(* PLC project Topicos, Desconocido Sin nombre 1 *)
(* stored: creationDateTime 2024-03-11T19:08:26, modificationDateTime 2024-03-26T02:22:43 *)

FUNCTION_BLOCK RedPetri
  VAR_EXTERNAL
    E_0 : BOOL;
    E_1 : BOOL;
    E_2 : BOOL;
    E_3 : BOOL;
    E_4 : BOOL;
    E_5 : BOOL;
    E_6 : BOOL;
    E_7 : BOOL;
    Start_Button : BOOL;
    Stop_Button : BOOL;
    Reset_Button : BOOL;
    Blue_Product_base_Sensor : BOOL;
    Green_Product_base_Sensor : BOOL;
    Metal_Product_base_Sensor : BOOL;
    Blue_Product_base_Sensor2 : BOOL;
    Green_Product_base_Sensor_2 : BOOL;
    Metal_Product_base_Sensor2 : BOOL;
    Blue_Product_Lid_Sensor : BOOL;
    Green_Product_Lid_Sensor : BOOL;
    Metal_Product_Lid_Sensor : BOOL;
    Blue_Item_Detected_Sensor : BOOL;
    Green_Item_Detected_Sensor : BOOL;
    Metal_Item_Detected_Sensor : BOOL;
    Blue_Item_Detected_Sensor_2 : BOOL;
    Green_Item_Detected_Sensor_2 : BOOL;
    Metal_Item_Detected_Sensor_2 : BOOL;
    Blue_Stackable_Box_Sensor : BOOL;
    Green_Stackable_Box_Sensor : BOOL;
    Metal_Stackable_Box_Sensor : BOOL;
    Blue_Rotate_sensor : BOOL;
    Green_Rotate_sensor : BOOL;
    Metal_Rotate_sensor : BOOL;
    Stacker_Crane_2_Moving_X : BOOL;
    Stacker_Crane_2_Moving_Z : BOOL;
    Stacker_Crane_3_Moving_X : BOOL;
    Stacker_Crane_3_Moving_Z : BOOL;
    Stacker_Crane_4_Moving_X : BOOL;
    Stacker_Crane_4_Moving_Z : BOOL;
    Turntable_GS_0_G_Sensor : BOOL;
    Turntable_GS_90_G_Sensor : BOOL;
    Turntable_GS_Back_Sensor : BOOL;
    Turntable_GS_Front_Sensor : BOOL;
    Turntable_MS_0_G_Sensor : BOOL;
    Turntable_MS_90_G_Sensor : BOOL;
    Turntable_MS_Back_Sensor : BOOL;
    Turntable_MS_Front_Sensor : BOOL;
    Sensor_Turntable_Blue_Station1 : BOOL;
    Sensor_Turntable_Green_Station1 : BOOL;
    Sensor_Turntable_Metal_Station1 : BOOL;
    Sensor_Turntable_Green_Station2 : BOOL;
    Sensor_Turntable_Metal_Station2 : BOOL;
    Stacker_Crane_2_Middle_Limit : BOOL;
    Stacker_Crane_3_Middle_Limit : BOOL;
    Stacker_Crane_4_Middle_Limit : BOOL;
    Stacker_Crane_2_Right_Limit : BOOL;
    Stacker_Crane_3_Right_Limit : BOOL;
    Stacker_Crane_4_Right_Limit : BOOL;
    Stacker_Crane_2_Left_Limit : BOOL;
    Stacker_Crane_3_Left_Limit : BOOL;
    Stacker_Crane_4_Left_Limit : BOOL;
    Start_Button_1_Light : BOOL;
    Stop_Button_1_Light : BOOL;
    Reset_Button_1_Light : BOOL;
    Blue_Sorter_Belt : BOOL;
    Green_Sorter_Belt : BOOL;
    Metal_Sorter_Belt : BOOL;
    Blue_Sorter_Turn : BOOL;
    Green_Sorter_Turn : BOOL;
    Metal_Sorter_Turn : BOOL;
    Belt_Conveyor_1 : BOOL;
    Belt_Conveyor_2 : BOOL;
    Blue_Belt_Conveyor_5 : BOOL;
    Blue_Belt_Conveyor_6 : BOOL;
    Blue_Belt_Conveyor_7 : BOOL;
    Blue_Belt_Conveyor_8 : BOOL;
    Green_Belt_Conveyor_5 : BOOL;
    Green_Belt_Conveyor_6 : BOOL;
    Green_Belt_Conveyor_7 : BOOL;
    Green_Belt_Conveyor_8 : BOOL;
    Metal_Belt_Conveyor_5 : BOOL;
    Metal_Belt_Conveyor_6 : BOOL;
    Metal_Belt_Conveyor_7 : BOOL;
    Metal_Belt_Conveyor_8 : BOOL;
    Blue_Positioner_1_Clamp : BOOL;
    Blue_Positioner_1_Raise : BOOL;
    Blue_Positioner_2_Clamp : BOOL;
    Blue_Positioner_1a_Clamp : BOOL;
    Green_Positioner_1_Clamp : BOOL;
    Green_Positioner_1_Raise : BOOL;
    Green_Positioner_2_Clamp : BOOL;
    Green_Positioner_1a_Clamp : BOOL;
    Metal_Positioner_1_Clamp : BOOL;
    Metal_Positioner_1_Raise : BOOL;
    Metal_Positioner_2_Clamp : BOOL;
    Metal_Positioner_1a_Clamp : BOOL;
    Blue_Pick_and_Place_Grab : BOOL;
    Blue_Pick_and_Place_Grab_2 : BOOL;
    Green_Pick_and_Place_Grab : BOOL;
    Green_Pick_and_Place_Grab_2 : BOOL;
    Metal_Pick_and_Place_Grab : BOOL;
    Metal_Pick_and_Place_Grab_2 : BOOL;
    Blue_Stackable_Box_Rotate : BOOL;
    Green_Stackable_Box_Rotate : BOOL;
    Metal_Stackable_Box_Rotate : BOOL;
    Blue_Pallet_Rotate : BOOL;
    Green_Pallet_Rotate : BOOL;
    Metal_Pallet_Rotate : BOOL;
    Stacker_Crane_2_Lift : BOOL;
    Stacker_Crane_3_Lift : BOOL;
    Stacker_Crane_4_Lift : BOOL;
    Stacker_Crane_2_Left : BOOL;
    Stacker_Crane_3_Left : BOOL;
    Stacker_Crane_4_Left : BOOL;
    Stacker_Crane_2_Right : BOOL;
    Stacker_Crane_3_Right : BOOL;
    Stacker_Crane_4_Right : BOOL;
    Turntable_GS_Roll_F : BOOL;
    Turntable_GS_Turn : BOOL;
    Turntable_MS_Roll_F : BOOL;
    Turntable_MS_Turn : BOOL;
    Loading_Conveyor_0 : BOOL;
    Loading_Conveyor_1 : BOOL;
    Loading_Conveyor_2 : BOOL;
    Loading_Conveyor_3 : BOOL;
    Loading_Conveyor_4 : BOOL;
    Blue_Belt_Conveyor_1 : BOOL;
    Blue_Belt_Conveyor_2 : BOOL;
    Blue_Belt_Conveyor_3 : BOOL;
    Blue_Belt_Conveyor_4 : BOOL;
    Green_Belt_Conveyor_1 : BOOL;
    Green_Belt_Conveyor_2 : BOOL;
    Green_Belt_Conveyor_3 : BOOL;
    Green_Belt_Conveyor_4 : BOOL;
    Metal_Belt_Conveyor_1 : BOOL;
    Curved_Roller_Conveyor_B : BOOL;
    Curved_Roller_Conveyor_F : BOOL;
    Roller_Conveyor_B2M : BOOL;
    Roller_Conveyor_M2G : BOOL;
    Roller_Conveyor_G2F : BOOL;
    Blue_Sensor : INT;
    Green_Sensor : INT;
    Metal_Sensor : INT;
    Blue_X_Position_Sensor : REAL;
    Blue_Z_Position_Sensor : REAL;
    Blue_X_Position_Sensor_2 : REAL;
    Blue_Z_Position_Sensor_2 : REAL;
    Green_X_Position_Sensor : REAL;
    Green_Z_Position_Sensor : REAL;
    Green_X_Position_Sensor_2 : REAL;
    Green_Z_Position_Sensor_2 : REAL;
    Metal_X_Position_Sensor : REAL;
    Metal_Z_Position_Sensor : REAL;
    Metal_X_Position_Sensor_2 : REAL;
    Metal_Z_Position_Sensor_2 : REAL;
    Blue_Sensor_2 : INT;
    Green_Sensor_2 : INT;
    Metal_Sensor2 : INT;
    Blue_Pick_and_Place_X_Set_Point : REAL;
    Blue_Pick_and_Place_Z_Set_Point : REAL;
    Blue_Pick_and_Place_X_Set_Point_2 : REAL;
    Blue_Pick_and_Place_Z_Set_Point_2 : REAL;
    Green_Pick_and_Place_X_Set_Point : REAL;
    Green_Pick_and_Place_Z_Set_Point : REAL;
    Green_Pick_and_Place_X_Set_Point_2 : REAL;
    Green_Pick_and_Place_Z_Set_Point_2 : REAL;
    Metal_Pick_and_Place_X_Set_Point : REAL;
    Metal_Pick_and_Place_Z_Set_Point : REAL;
    Metal_Pick_and_Place_X_Set_Point_2 : REAL;
    Metal_Pick_and_Place_Z_Set_Point_2 : REAL;
    Stacker_Crane_2_Target_Position : INT;
    Stacker_Crane_3_Target_Position : INT;
    Stacker_Crane_4_Target_Position : INT;
  END_VAR

            If E_0 = True Then



      E_0 := False;

      E_1 := True;



  End_If;
          
END_FUNCTION_BLOCK

FUNCTION_BLOCK Actuadores
  VAR_EXTERNAL
    E_0 : BOOL;
    E_1 : BOOL;
    E_2 : BOOL;
    E_3 : BOOL;
    E_4 : BOOL;
    E_5 : BOOL;
    E_6 : BOOL;
    E_7 : BOOL;
    Start_Button : BOOL;
    Stop_Button : BOOL;
    Reset_Button : BOOL;
    Blue_Product_base_Sensor : BOOL;
    Green_Product_base_Sensor : BOOL;
    Metal_Product_base_Sensor : BOOL;
    Blue_Product_base_Sensor2 : BOOL;
    Green_Product_base_Sensor_2 : BOOL;
    Metal_Product_base_Sensor2 : BOOL;
    Blue_Product_Lid_Sensor : BOOL;
    Green_Product_Lid_Sensor : BOOL;
    Metal_Product_Lid_Sensor : BOOL;
    Blue_Item_Detected_Sensor : BOOL;
    Green_Item_Detected_Sensor : BOOL;
    Metal_Item_Detected_Sensor : BOOL;
    Blue_Item_Detected_Sensor_2 : BOOL;
    Green_Item_Detected_Sensor_2 : BOOL;
    Metal_Item_Detected_Sensor_2 : BOOL;
    Blue_Stackable_Box_Sensor : BOOL;
    Green_Stackable_Box_Sensor : BOOL;
    Metal_Stackable_Box_Sensor : BOOL;
    Blue_Rotate_sensor : BOOL;
    Green_Rotate_sensor : BOOL;
    Metal_Rotate_sensor : BOOL;
    Stacker_Crane_2_Moving_X : BOOL;
    Stacker_Crane_2_Moving_Z : BOOL;
    Stacker_Crane_3_Moving_X : BOOL;
    Stacker_Crane_3_Moving_Z : BOOL;
    Stacker_Crane_4_Moving_X : BOOL;
    Stacker_Crane_4_Moving_Z : BOOL;
    Turntable_GS_0_G_Sensor : BOOL;
    Turntable_GS_90_G_Sensor : BOOL;
    Turntable_GS_Back_Sensor : BOOL;
    Turntable_GS_Front_Sensor : BOOL;
    Turntable_MS_0_G_Sensor : BOOL;
    Turntable_MS_90_G_Sensor : BOOL;
    Turntable_MS_Back_Sensor : BOOL;
    Turntable_MS_Front_Sensor : BOOL;
    Sensor_Turntable_Blue_Station1 : BOOL;
    Sensor_Turntable_Green_Station1 : BOOL;
    Sensor_Turntable_Metal_Station1 : BOOL;
    Sensor_Turntable_Green_Station2 : BOOL;
    Sensor_Turntable_Metal_Station2 : BOOL;
    Stacker_Crane_2_Middle_Limit : BOOL;
    Stacker_Crane_3_Middle_Limit : BOOL;
    Stacker_Crane_4_Middle_Limit : BOOL;
    Stacker_Crane_2_Right_Limit : BOOL;
    Stacker_Crane_3_Right_Limit : BOOL;
    Stacker_Crane_4_Right_Limit : BOOL;
    Stacker_Crane_2_Left_Limit : BOOL;
    Stacker_Crane_3_Left_Limit : BOOL;
    Stacker_Crane_4_Left_Limit : BOOL;
    Start_Button_1_Light : BOOL;
    Stop_Button_1_Light : BOOL;
    Reset_Button_1_Light : BOOL;
    Blue_Sorter_Belt : BOOL;
    Green_Sorter_Belt : BOOL;
    Metal_Sorter_Belt : BOOL;
    Blue_Sorter_Turn : BOOL;
    Green_Sorter_Turn : BOOL;
    Metal_Sorter_Turn : BOOL;
    Belt_Conveyor_1 : BOOL;
    Belt_Conveyor_2 : BOOL;
    Blue_Belt_Conveyor_5 : BOOL;
    Blue_Belt_Conveyor_6 : BOOL;
    Blue_Belt_Conveyor_7 : BOOL;
    Blue_Belt_Conveyor_8 : BOOL;
    Green_Belt_Conveyor_5 : BOOL;
    Green_Belt_Conveyor_6 : BOOL;
    Green_Belt_Conveyor_7 : BOOL;
    Green_Belt_Conveyor_8 : BOOL;
    Metal_Belt_Conveyor_5 : BOOL;
    Metal_Belt_Conveyor_6 : BOOL;
    Metal_Belt_Conveyor_7 : BOOL;
    Metal_Belt_Conveyor_8 : BOOL;
    Blue_Positioner_1_Clamp : BOOL;
    Blue_Positioner_1_Raise : BOOL;
    Blue_Positioner_2_Clamp : BOOL;
    Blue_Positioner_1a_Clamp : BOOL;
    Green_Positioner_1_Clamp : BOOL;
    Green_Positioner_1_Raise : BOOL;
    Green_Positioner_2_Clamp : BOOL;
    Green_Positioner_1a_Clamp : BOOL;
    Metal_Positioner_1_Clamp : BOOL;
    Metal_Positioner_1_Raise : BOOL;
    Metal_Positioner_2_Clamp : BOOL;
    Metal_Positioner_1a_Clamp : BOOL;
    Blue_Pick_and_Place_Grab : BOOL;
    Blue_Pick_and_Place_Grab_2 : BOOL;
    Green_Pick_and_Place_Grab : BOOL;
    Green_Pick_and_Place_Grab_2 : BOOL;
    Metal_Pick_and_Place_Grab : BOOL;
    Metal_Pick_and_Place_Grab_2 : BOOL;
    Blue_Stackable_Box_Rotate : BOOL;
    Green_Stackable_Box_Rotate : BOOL;
    Metal_Stackable_Box_Rotate : BOOL;
    Blue_Pallet_Rotate : BOOL;
    Green_Pallet_Rotate : BOOL;
    Metal_Pallet_Rotate : BOOL;
    Stacker_Crane_2_Lift : BOOL;
    Stacker_Crane_3_Lift : BOOL;
    Stacker_Crane_4_Lift : BOOL;
    Stacker_Crane_2_Left : BOOL;
    Stacker_Crane_3_Left : BOOL;
    Stacker_Crane_4_Left : BOOL;
    Stacker_Crane_2_Right : BOOL;
    Stacker_Crane_3_Right : BOOL;
    Stacker_Crane_4_Right : BOOL;
    Turntable_GS_Roll_F : BOOL;
    Turntable_GS_Turn : BOOL;
    Turntable_MS_Roll_F : BOOL;
    Turntable_MS_Turn : BOOL;
    Loading_Conveyor_0 : BOOL;
    Loading_Conveyor_1 : BOOL;
    Loading_Conveyor_2 : BOOL;
    Loading_Conveyor_3 : BOOL;
    Loading_Conveyor_4 : BOOL;
    Blue_Belt_Conveyor_1 : BOOL;
    Blue_Belt_Conveyor_2 : BOOL;
    Blue_Belt_Conveyor_3 : BOOL;
    Blue_Belt_Conveyor_4 : BOOL;
    Green_Belt_Conveyor_1 : BOOL;
    Green_Belt_Conveyor_2 : BOOL;
    Green_Belt_Conveyor_3 : BOOL;
    Green_Belt_Conveyor_4 : BOOL;
    Metal_Belt_Conveyor_1 : BOOL;
    Curved_Roller_Conveyor_B : BOOL;
    Curved_Roller_Conveyor_F : BOOL;
    Roller_Conveyor_B2M : BOOL;
    Roller_Conveyor_M2G : BOOL;
    Roller_Conveyor_G2F : BOOL;
    Blue_Sensor : INT;
    Green_Sensor : INT;
    Metal_Sensor : INT;
    Blue_X_Position_Sensor : REAL;
    Blue_Z_Position_Sensor : REAL;
    Blue_X_Position_Sensor_2 : REAL;
    Blue_Z_Position_Sensor_2 : REAL;
    Green_X_Position_Sensor : REAL;
    Green_Z_Position_Sensor : REAL;
    Green_X_Position_Sensor_2 : REAL;
    Green_Z_Position_Sensor_2 : REAL;
    Metal_X_Position_Sensor : REAL;
    Metal_Z_Position_Sensor : REAL;
    Metal_X_Position_Sensor_2 : REAL;
    Metal_Z_Position_Sensor_2 : REAL;
    Blue_Sensor_2 : INT;
    Green_Sensor_2 : INT;
    Metal_Sensor2 : INT;
    Blue_Pick_and_Place_X_Set_Point : REAL;
    Blue_Pick_and_Place_Z_Set_Point : REAL;
    Blue_Pick_and_Place_X_Set_Point_2 : REAL;
    Blue_Pick_and_Place_Z_Set_Point_2 : REAL;
    Green_Pick_and_Place_X_Set_Point : REAL;
    Green_Pick_and_Place_Z_Set_Point : REAL;
    Green_Pick_and_Place_X_Set_Point_2 : REAL;
    Green_Pick_and_Place_Z_Set_Point_2 : REAL;
    Metal_Pick_and_Place_X_Set_Point : REAL;
    Metal_Pick_and_Place_Z_Set_Point : REAL;
    Metal_Pick_and_Place_X_Set_Point_2 : REAL;
    Metal_Pick_and_Place_Z_Set_Point_2 : REAL;
    Stacker_Crane_2_Target_Position : INT;
    Stacker_Crane_3_Target_Position : INT;
    Stacker_Crane_4_Target_Position : INT;
  END_VAR

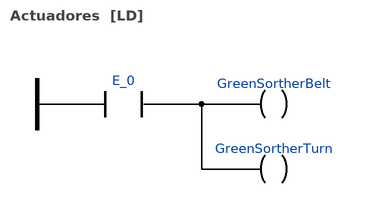
(* LD diagram, written out as Structured Text *)
GreenSortherBelt := E_0;
GreenSortherTurn := E_0;
END_FUNCTION_BLOCK

PROGRAM OB1
  VAR_EXTERNAL
    E_0 : BOOL;
    E_1 : BOOL;
    E_2 : BOOL;
    E_3 : BOOL;
    E_4 : BOOL;
    E_5 : BOOL;
    E_6 : BOOL;
    E_7 : BOOL;
    Start_Button : BOOL;
    Stop_Button : BOOL;
    Reset_Button : BOOL;
    Blue_Product_base_Sensor : BOOL;
    Green_Product_base_Sensor : BOOL;
    Metal_Product_base_Sensor : BOOL;
    Blue_Product_base_Sensor2 : BOOL;
    Green_Product_base_Sensor_2 : BOOL;
    Metal_Product_base_Sensor2 : BOOL;
    Blue_Product_Lid_Sensor : BOOL;
    Green_Product_Lid_Sensor : BOOL;
    Metal_Product_Lid_Sensor : BOOL;
    Blue_Item_Detected_Sensor : BOOL;
    Green_Item_Detected_Sensor : BOOL;
    Metal_Item_Detected_Sensor : BOOL;
    Blue_Item_Detected_Sensor_2 : BOOL;
    Green_Item_Detected_Sensor_2 : BOOL;
    Metal_Item_Detected_Sensor_2 : BOOL;
    Blue_Stackable_Box_Sensor : BOOL;
    Green_Stackable_Box_Sensor : BOOL;
    Metal_Stackable_Box_Sensor : BOOL;
    Blue_Rotate_sensor : BOOL;
    Green_Rotate_sensor : BOOL;
    Metal_Rotate_sensor : BOOL;
    Stacker_Crane_2_Moving_X : BOOL;
    Stacker_Crane_2_Moving_Z : BOOL;
    Stacker_Crane_3_Moving_X : BOOL;
    Stacker_Crane_3_Moving_Z : BOOL;
    Stacker_Crane_4_Moving_X : BOOL;
    Stacker_Crane_4_Moving_Z : BOOL;
    Turntable_GS_0_G_Sensor : BOOL;
    Turntable_GS_90_G_Sensor : BOOL;
    Turntable_GS_Back_Sensor : BOOL;
    Turntable_GS_Front_Sensor : BOOL;
    Turntable_MS_0_G_Sensor : BOOL;
    Turntable_MS_90_G_Sensor : BOOL;
    Turntable_MS_Back_Sensor : BOOL;
    Turntable_MS_Front_Sensor : BOOL;
    Sensor_Turntable_Blue_Station1 : BOOL;
    Sensor_Turntable_Green_Station1 : BOOL;
    Sensor_Turntable_Metal_Station1 : BOOL;
    Sensor_Turntable_Green_Station2 : BOOL;
    Sensor_Turntable_Metal_Station2 : BOOL;
    Stacker_Crane_2_Middle_Limit : BOOL;
    Stacker_Crane_3_Middle_Limit : BOOL;
    Stacker_Crane_4_Middle_Limit : BOOL;
    Stacker_Crane_2_Right_Limit : BOOL;
    Stacker_Crane_3_Right_Limit : BOOL;
    Stacker_Crane_4_Right_Limit : BOOL;
    Stacker_Crane_2_Left_Limit : BOOL;
    Stacker_Crane_3_Left_Limit : BOOL;
    Stacker_Crane_4_Left_Limit : BOOL;
    Start_Button_1_Light : BOOL;
    Stop_Button_1_Light : BOOL;
    Reset_Button_1_Light : BOOL;
    Blue_Sorter_Belt : BOOL;
    Green_Sorter_Belt : BOOL;
    Metal_Sorter_Belt : BOOL;
    Blue_Sorter_Turn : BOOL;
    Green_Sorter_Turn : BOOL;
    Metal_Sorter_Turn : BOOL;
    Belt_Conveyor_1 : BOOL;
    Belt_Conveyor_2 : BOOL;
    Blue_Belt_Conveyor_5 : BOOL;
    Blue_Belt_Conveyor_6 : BOOL;
    Blue_Belt_Conveyor_7 : BOOL;
    Blue_Belt_Conveyor_8 : BOOL;
    Green_Belt_Conveyor_5 : BOOL;
    Green_Belt_Conveyor_6 : BOOL;
    Green_Belt_Conveyor_7 : BOOL;
    Green_Belt_Conveyor_8 : BOOL;
    Metal_Belt_Conveyor_5 : BOOL;
    Metal_Belt_Conveyor_6 : BOOL;
    Metal_Belt_Conveyor_7 : BOOL;
    Metal_Belt_Conveyor_8 : BOOL;
    Blue_Positioner_1_Clamp : BOOL;
    Blue_Positioner_1_Raise : BOOL;
    Blue_Positioner_2_Clamp : BOOL;
    Blue_Positioner_1a_Clamp : BOOL;
    Green_Positioner_1_Clamp : BOOL;
    Green_Positioner_1_Raise : BOOL;
    Green_Positioner_2_Clamp : BOOL;
    Green_Positioner_1a_Clamp : BOOL;
    Metal_Positioner_1_Clamp : BOOL;
    Metal_Positioner_1_Raise : BOOL;
    Metal_Positioner_2_Clamp : BOOL;
    Metal_Positioner_1a_Clamp : BOOL;
    Blue_Pick_and_Place_Grab : BOOL;
    Blue_Pick_and_Place_Grab_2 : BOOL;
    Green_Pick_and_Place_Grab : BOOL;
    Green_Pick_and_Place_Grab_2 : BOOL;
    Metal_Pick_and_Place_Grab : BOOL;
    Metal_Pick_and_Place_Grab_2 : BOOL;
    Blue_Stackable_Box_Rotate : BOOL;
    Green_Stackable_Box_Rotate : BOOL;
    Metal_Stackable_Box_Rotate : BOOL;
    Blue_Pallet_Rotate : BOOL;
    Green_Pallet_Rotate : BOOL;
    Metal_Pallet_Rotate : BOOL;
    Stacker_Crane_2_Lift : BOOL;
    Stacker_Crane_3_Lift : BOOL;
    Stacker_Crane_4_Lift : BOOL;
    Stacker_Crane_2_Left : BOOL;
    Stacker_Crane_3_Left : BOOL;
    Stacker_Crane_4_Left : BOOL;
    Stacker_Crane_2_Right : BOOL;
    Stacker_Crane_3_Right : BOOL;
    Stacker_Crane_4_Right : BOOL;
    Turntable_GS_Roll_F : BOOL;
    Turntable_GS_Turn : BOOL;
    Turntable_MS_Roll_F : BOOL;
    Turntable_MS_Turn : BOOL;
    Loading_Conveyor_0 : BOOL;
    Loading_Conveyor_1 : BOOL;
    Loading_Conveyor_2 : BOOL;
    Loading_Conveyor_3 : BOOL;
    Loading_Conveyor_4 : BOOL;
    Blue_Belt_Conveyor_1 : BOOL;
    Blue_Belt_Conveyor_2 : BOOL;
    Blue_Belt_Conveyor_3 : BOOL;
    Blue_Belt_Conveyor_4 : BOOL;
    Green_Belt_Conveyor_1 : BOOL;
    Green_Belt_Conveyor_2 : BOOL;
    Green_Belt_Conveyor_3 : BOOL;
    Green_Belt_Conveyor_4 : BOOL;
    Metal_Belt_Conveyor_1 : BOOL;
    Curved_Roller_Conveyor_B : BOOL;
    Curved_Roller_Conveyor_F : BOOL;
    Roller_Conveyor_B2M : BOOL;
    Roller_Conveyor_M2G : BOOL;
    Roller_Conveyor_G2F : BOOL;
    Blue_Sensor : INT;
    Green_Sensor : INT;
    Metal_Sensor : INT;
    Blue_X_Position_Sensor : REAL;
    Blue_Z_Position_Sensor : REAL;
    Blue_X_Position_Sensor_2 : REAL;
    Blue_Z_Position_Sensor_2 : REAL;
    Green_X_Position_Sensor : REAL;
    Green_Z_Position_Sensor : REAL;
    Green_X_Position_Sensor_2 : REAL;
    Green_Z_Position_Sensor_2 : REAL;
    Metal_X_Position_Sensor : REAL;
    Metal_Z_Position_Sensor : REAL;
    Metal_X_Position_Sensor_2 : REAL;
    Metal_Z_Position_Sensor_2 : REAL;
    Blue_Sensor_2 : INT;
    Green_Sensor_2 : INT;
    Metal_Sensor2 : INT;
    Blue_Pick_and_Place_X_Set_Point : REAL;
    Blue_Pick_and_Place_Z_Set_Point : REAL;
    Blue_Pick_and_Place_X_Set_Point_2 : REAL;
    Blue_Pick_and_Place_Z_Set_Point_2 : REAL;
    Green_Pick_and_Place_X_Set_Point : REAL;
    Green_Pick_and_Place_Z_Set_Point : REAL;
    Green_Pick_and_Place_X_Set_Point_2 : REAL;
    Green_Pick_and_Place_Z_Set_Point_2 : REAL;
    Metal_Pick_and_Place_X_Set_Point : REAL;
    Metal_Pick_and_Place_Z_Set_Point : REAL;
    Metal_Pick_and_Place_X_Set_Point_2 : REAL;
    Metal_Pick_and_Place_Z_Set_Point_2 : REAL;
    Stacker_Crane_2_Target_Position : INT;
    Stacker_Crane_3_Target_Position : INT;
    Stacker_Crane_4_Target_Position : INT;
  END_VAR
  VAR
    RedPetri0 : RedPetri;
    Actuadores0 : Actuadores;
  END_VAR

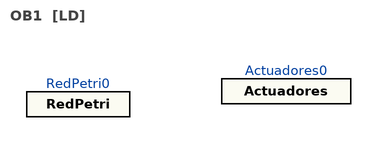
(* LD diagram, written out as Structured Text *)
Actuadores0();
RedPetri0();
END_PROGRAM

CONFIGURATION Config0
  RESOURCE Res0 ON PLC
    VAR_GLOBAL
      E_0 : BOOL := True;
      E_1 : BOOL := False;
      E_2 : BOOL := False;
      E_3 : BOOL := False;
      E_4 : BOOL := False;
      E_5 : BOOL := False;
      E_6 : BOOL := False;
      E_7 : BOOL := False;
      Start_Button AT %IX100.0 : BOOL := False;
      Stop_Button AT %IX100.1 : BOOL := False;
      Reset_Button AT %IX100.2 : BOOL := False;
      Blue_Product_base_Sensor AT %IX100.3 : BOOL := False;
      Green_Product_base_Sensor AT %IX100.4 : BOOL := False;
      Metal_Product_base_Sensor AT %IX100.5 : BOOL := False;
      Blue_Product_base_Sensor2 AT %IX100.6 : BOOL := False;
      Green_Product_base_Sensor_2 AT %IX100.7 : BOOL := False;
      Metal_Product_base_Sensor2 AT %IX100.8 : BOOL := False;
      Blue_Product_Lid_Sensor AT %IX100.9 : BOOL := False;
      Green_Product_Lid_Sensor AT %IX100.10 : BOOL := False;
      Metal_Product_Lid_Sensor AT %IX100.11 : BOOL := False;
      Blue_Item_Detected_Sensor AT %IX100.12 : BOOL := False;
      Green_Item_Detected_Sensor AT %IX100.13 : BOOL := False;
      Metal_Item_Detected_Sensor AT %IX100.14 : BOOL := False;
      Blue_Item_Detected_Sensor_2 AT %IX100.15 : BOOL := False;
      Green_Item_Detected_Sensor_2 AT %IX100.16 : BOOL := False;
      Metal_Item_Detected_Sensor_2 AT %IX100.17 : BOOL := False;
      Blue_Stackable_Box_Sensor AT %IX100.18 : BOOL := False;
      Green_Stackable_Box_Sensor AT %IX100.19 : BOOL := False;
      Metal_Stackable_Box_Sensor AT %IX100.20 : BOOL := False;
      Blue_Rotate_sensor AT %IX100.21 : BOOL := False;
      Green_Rotate_sensor AT %IX100.22 : BOOL := False;
      Metal_Rotate_sensor AT %IX100.23 : BOOL := False;
      Stacker_Crane_2_Moving_X AT %IX100.24 : BOOL := False;
      Stacker_Crane_2_Moving_Z AT %IX100.25 : BOOL := False;
      Stacker_Crane_3_Moving_X AT %IX100.26 : BOOL := False;
      Stacker_Crane_3_Moving_Z AT %IX100.27 : BOOL := False;
      Stacker_Crane_4_Moving_X AT %IX100.28 : BOOL := False;
      Stacker_Crane_4_Moving_Z AT %IX100.29 : BOOL := False;
      Turntable_GS_0_G_Sensor AT %IX100.30 : BOOL := False;
      Turntable_GS_90_G_Sensor AT %IX100.31 : BOOL := False;
      Turntable_GS_Back_Sensor AT %IX100.32 : BOOL := False;
      Turntable_GS_Front_Sensor AT %IX100.33 : BOOL := False;
      Turntable_MS_0_G_Sensor AT %IX100.34 : BOOL := False;
      Turntable_MS_90_G_Sensor AT %IX100.35 : BOOL := False;
      Turntable_MS_Back_Sensor AT %IX100.36 : BOOL := False;
      Turntable_MS_Front_Sensor AT %IX100.37 : BOOL := False;
      Sensor_Turntable_Blue_Station1 AT %IX100.38 : BOOL := False;
      Sensor_Turntable_Green_Station1 AT %IX100.39 : BOOL := False;
      Sensor_Turntable_Metal_Station1 AT %IX100.40 : BOOL := False;
      Sensor_Turntable_Green_Station2 AT %IX100.41 : BOOL := False;
      Sensor_Turntable_Metal_Station2 AT %IX100.42 : BOOL := False;
      Stacker_Crane_2_Middle_Limit AT %IX100.43 : BOOL := False;
      Stacker_Crane_3_Middle_Limit AT %IX100.44 : BOOL := False;
      Stacker_Crane_4_Middle_Limit AT %IX100.45 : BOOL := False;
      Stacker_Crane_2_Right_Limit AT %IX100.46 : BOOL := False;
      Stacker_Crane_3_Right_Limit AT %IX100.47 : BOOL := False;
      Stacker_Crane_4_Right_Limit AT %IX100.48 : BOOL := False;
      Stacker_Crane_2_Left_Limit AT %IX100.49 : BOOL := False;
      Stacker_Crane_3_Left_Limit AT %IX100.50 : BOOL := False;
      Stacker_Crane_4_Left_Limit AT %IX100.51 : BOOL := False;
      Start_Button_1_Light AT %QX100.0 : BOOL := False;
      Stop_Button_1_Light AT %QX100.1 : BOOL := False;
      Reset_Button_1_Light AT %QX100.2 : BOOL := False;
      Blue_Sorter_Belt AT %QX100.3 : BOOL := False;
      Green_Sorter_Belt AT %QX100.4 : BOOL := False;
      Metal_Sorter_Belt AT %QX100.5 : BOOL := False;
      Blue_Sorter_Turn AT %QX100.6 : BOOL := False;
      Green_Sorter_Turn AT %QX100.7 : BOOL := False;
      Metal_Sorter_Turn AT %QX100.8 : BOOL := False;
      Belt_Conveyor_1 AT %QX100.9 : BOOL := False;
      Belt_Conveyor_2 AT %QX100.10 : BOOL := False;
      Blue_Belt_Conveyor_5 AT %QX100.11 : BOOL := False;
      Blue_Belt_Conveyor_6 AT %QX100.12 : BOOL := False;
      Blue_Belt_Conveyor_7 AT %QX100.13 : BOOL := False;
      Blue_Belt_Conveyor_8 AT %QX100.14 : BOOL := False;
      Green_Belt_Conveyor_5 AT %QX100.15 : BOOL := False;
      Green_Belt_Conveyor_6 AT %QX100.16 : BOOL := False;
      Green_Belt_Conveyor_7 AT %QX100.17 : BOOL := False;
      Green_Belt_Conveyor_8 AT %QX100.18 : BOOL := False;
      Metal_Belt_Conveyor_5 AT %QX100.19 : BOOL := False;
      Metal_Belt_Conveyor_6 AT %QX100.20 : BOOL := False;
      Metal_Belt_Conveyor_7 AT %QX100.21 : BOOL := False;
      Metal_Belt_Conveyor_8 AT %QX100.22 : BOOL := False;
      Blue_Positioner_1_Clamp AT %QX100.23 : BOOL := False;
      Blue_Positioner_1_Raise AT %QX100.24 : BOOL := False;
      Blue_Positioner_2_Clamp AT %QX100.25 : BOOL := False;
      Blue_Positioner_1a_Clamp AT %QX100.26 : BOOL := False;
      Green_Positioner_1_Clamp AT %QX100.27 : BOOL := False;
      Green_Positioner_1_Raise AT %QX100.28 : BOOL := False;
      Green_Positioner_2_Clamp AT %QX100.29 : BOOL := False;
      Green_Positioner_1a_Clamp AT %QX100.30 : BOOL := False;
      Metal_Positioner_1_Clamp AT %QX100.31 : BOOL := False;
      Metal_Positioner_1_Raise AT %QX100.32 : BOOL := False;
      Metal_Positioner_2_Clamp AT %QX100.33 : BOOL := False;
      Metal_Positioner_1a_Clamp AT %QX100.34 : BOOL := False;
      Blue_Pick_and_Place_Grab AT %QX100.35 : BOOL := False;
      Blue_Pick_and_Place_Grab_2 AT %QX100.36 : BOOL := False;
      Green_Pick_and_Place_Grab AT %QX100.37 : BOOL := False;
      Green_Pick_and_Place_Grab_2 AT %QX100.38 : BOOL := False;
      Metal_Pick_and_Place_Grab AT %QX100.39 : BOOL := False;
      Metal_Pick_and_Place_Grab_2 AT %QX100.40 : BOOL := False;
      Blue_Stackable_Box_Rotate AT %QX100.41 : BOOL := False;
      Green_Stackable_Box_Rotate AT %QX100.42 : BOOL := False;
      Metal_Stackable_Box_Rotate AT %QX100.43 : BOOL := False;
      Blue_Pallet_Rotate AT %QX100.44 : BOOL := False;
      Green_Pallet_Rotate AT %QX100.45 : BOOL := False;
      Metal_Pallet_Rotate AT %QX100.46 : BOOL := False;
      Stacker_Crane_2_Lift AT %QX100.47 : BOOL := False;
      Stacker_Crane_3_Lift AT %QX100.48 : BOOL := False;
      Stacker_Crane_4_Lift AT %QX100.49 : BOOL := False;
      Stacker_Crane_2_Left AT %QX100.50 : BOOL := False;
      Stacker_Crane_3_Left AT %QX100.51 : BOOL := False;
      Stacker_Crane_4_Left AT %QX100.52 : BOOL := False;
      Stacker_Crane_2_Right AT %QX100.53 : BOOL := False;
      Stacker_Crane_3_Right AT %QX100.54 : BOOL := False;
      Stacker_Crane_4_Right AT %QX100.55 : BOOL := False;
      Turntable_GS_Roll_F AT %QX100.56 : BOOL := False;
      Turntable_GS_Turn AT %QX100.57 : BOOL := False;
      Turntable_MS_Roll_F AT %QX100.58 : BOOL := False;
      Turntable_MS_Turn AT %QX100.59 : BOOL := False;
      Loading_Conveyor_0 AT %QX100.60 : BOOL := False;
      Loading_Conveyor_1 AT %QX100.61 : BOOL := False;
      Loading_Conveyor_2 AT %QX100.62 : BOOL := False;
      Loading_Conveyor_3 AT %QX100.63 : BOOL := False;
      Loading_Conveyor_4 AT %QX100.64 : BOOL := False;
      Blue_Belt_Conveyor_1 AT %QX100.65 : BOOL := False;
      Blue_Belt_Conveyor_2 AT %QX100.66 : BOOL := False;
      Blue_Belt_Conveyor_3 AT %QX100.67 : BOOL := False;
      Blue_Belt_Conveyor_4 AT %QX100.68 : BOOL := False;
      Green_Belt_Conveyor_1 AT %QX100.69 : BOOL := False;
      Green_Belt_Conveyor_2 AT %QX100.70 : BOOL := False;
      Green_Belt_Conveyor_3 AT %QX100.71 : BOOL := False;
      Green_Belt_Conveyor_4 AT %QX100.72 : BOOL := False;
      Metal_Belt_Conveyor_1 AT %QX100.73 : BOOL := False;
      Curved_Roller_Conveyor_B AT %QX100.74 : BOOL := False;
      Curved_Roller_Conveyor_F AT %QX100.75 : BOOL := False;
      Roller_Conveyor_B2M AT %QX100.76 : BOOL := False;
      Roller_Conveyor_M2G AT %QX100.77 : BOOL := False;
      Roller_Conveyor_G2F AT %QX100.78 : BOOL := False;
      Blue_Sensor AT %IW100 : INT := 0;
      Green_Sensor AT %IW101 : INT := 0;
      Metal_Sensor AT %IW102 : INT := 0;
      Blue_X_Position_Sensor AT %IW103 : REAL := 0;
      Blue_Z_Position_Sensor AT %IW104 : REAL := 0;
      Blue_X_Position_Sensor_2 AT %IW105 : REAL := 0;
      Blue_Z_Position_Sensor_2 AT %IW106 : REAL := 0;
      Green_X_Position_Sensor AT %IW107 : REAL := 0;
      Green_Z_Position_Sensor AT %IW108 : REAL := 0;
      Green_X_Position_Sensor_2 AT %IW109 : REAL := 0;
      Green_Z_Position_Sensor_2 AT %IW110 : REAL := 0;
      Metal_X_Position_Sensor AT %IW111 : REAL := 0;
      Metal_Z_Position_Sensor AT %IW112 : REAL := 0;
      Metal_X_Position_Sensor_2 AT %IW113 : REAL := 0;
      Metal_Z_Position_Sensor_2 AT %IW114 : REAL := 0;
      Blue_Sensor_2 AT %IW115 : INT := 0;
      Green_Sensor_2 AT %IW116 : INT := 0;
      Metal_Sensor2 AT %IW117 : INT := 0;
      Blue_Pick_and_Place_X_Set_Point AT %QW100 : REAL := 0;
      Blue_Pick_and_Place_Z_Set_Point AT %QW101 : REAL := 0;
      Blue_Pick_and_Place_X_Set_Point_2 AT %QW102 : REAL := 0;
      Blue_Pick_and_Place_Z_Set_Point_2 AT %QW103 : REAL := 0;
      Green_Pick_and_Place_X_Set_Point AT %QW104 : REAL := 0;
      Green_Pick_and_Place_Z_Set_Point AT %QW105 : REAL := 0;
      Green_Pick_and_Place_X_Set_Point_2 AT %QW106 : REAL := 0;
      Green_Pick_and_Place_Z_Set_Point_2 AT %QW107 : REAL := 0;
      Metal_Pick_and_Place_X_Set_Point AT %QW108 : REAL := 0;
      Metal_Pick_and_Place_Z_Set_Point AT %QW109 : REAL := 0;
      Metal_Pick_and_Place_X_Set_Point_2 AT %QW110 : REAL := 0;
      Metal_Pick_and_Place_Z_Set_Point_2 AT %QW111 : REAL := 0;
      Stacker_Crane_2_Target_Position AT %QW115 : INT := 0;
      Stacker_Crane_3_Target_Position AT %QW116 : INT := 0;
      Stacker_Crane_4_Target_Position AT %QW117 : INT := 0;
    END_VAR
    TASK task0(INTERVAL := T#20ms, PRIORITY := 0);
    PROGRAM instance0 WITH task0 : OB1;
  END_RESOURCE
END_CONFIGURATION
